Fanuc KAREL source: kb00127.KL

PROGRAM KB00127
%STACKSIZE=65535
%PRIORITY=65535
%NOLOCKGROUP
VAR
P1 : STRING[80]
P2 : INTEGER
RESULT : INTEGER
BEGIN
P1='A'
P2=1
-- UNRESOLVED_PC line 10 opcodes [27 22 2A 22 76 23] marker_code=26
END KB00127
